(* IEC 61131-3 sources: HappyLearnCodesys/content/softmotion/BasicMotion_DigitalCamSwitch_HighPrecision, 11 files *)

(* ---- GVL_EL2252.st ---- *)
{attribute 'qualified_only'}
VAR_GLOBAL CONSTANT
    /// Maximum number of channels for the EL2252
    NUM_CHANNELS : UDINT := 2;
END_VAR

(* ---- GVL_GVL_EL2252.st ---- *)
END_VAR
{attribute 'qualified_only'}
VAR_GLOBAL CONSTANT
NUM_CHANNELS : UDINT := 2;
/// Maximum number of channels for the EL2252

(* ---- DurationTo32bitEtcTimestamp.st ---- *)
/// Converts duration in seconds to 32bit EtherCAT timestamp in nanoseconds.
FUNCTION DurationTo32bitEtcTimestamp : UDINT
VAR_IN_OUT
    Axis : AXIS_REF_SM3;
	ETCMaster : IODrvEtherCAT;
END_VAR
VAR_INPUT
    duration : LREAL;
END_VAR
VAR
    timestamp64Bit : ULINT;
END_VAR

timestamp64Bit := DurationTo64bitEtcTimestamp(Axis, ETCMaster, duration);
DurationTo32bitEtcTimestamp := TO_UDINT(timestamp64Bit AND 16#FFFF_FFFF);

(* ---- DurationTo64bitEtcTimestamp.st ---- *)
/// Converts duration in seconds to 64bit EtherCAT timestamp in nanoseconds.
FUNCTION DurationTo64bitEtcTimestamp : ULINT
VAR_IN_OUT
    Axis : AXIS_REF_SM3;
	ETCMaster : IODrvEtherCAT;
END_VAR
VAR_INPUT
    duration : LREAL;
END_VAR
VAR
    curTime_ns : ULINT;
	error : SMC_ERROR ;
END_VAR

{IF defined (pou: AXIS_REF_SM3.GetTimestampActValues)}
// GetTimeStampActValues exists for SoftMotion version 4.19.0.0 and higher.
error := Axis.GetTimestampActValues(CurrentActTime=> curTime_ns);
IF error = SMC_NOT_IMPLEMENTED THEN
	// No EtherCAT drive, fall back to default implementation
	curTime_ns := ETCMaster.DCClockReferenceTime;
END_IF
{ELSE}
curTime_ns := ETCMaster.DCClockReferenceTime;
{END_IF}
DurationTo64bitEtcTimestamp := curTime_ns + TO_ULINT(duration*1E9);

(* ---- EventId_GreaterThan.st ---- *)
/// Returns whether the given event Id id1 is greater than the event Id id2.
/// Note that if id2 is not valid, id1 is considered greater.
FUNCTION EventId_GreaterThan : BOOL
VAR_INPUT
    id1 : UDINT;
END_VAR
VAR_IN_OUT CONSTANT
    id2 : EventId;
END_VAR

IF NOT id2.valid THEN
    EventId_GreaterThan := TRUE;
ELSE
    // Greater than check with handling of 32-bit overflows
    EventId_GreaterThan :=
        (id1 > id2.id AND id1 - id2.id < 16#7FFF_FFFF) OR_ELSE
        (id1 < id2.id AND id2.id - id1 > 16#7FFF_FFFF);
END_IF

(* ---- EventId_Init.st ---- *)
FUNCTION EventId_Init
VAR_IN_OUT
    lte : EventId;
END_VAR

lte.id := 0;
lte.valid := FALSE;

(* ---- EventId_Set.st ---- *)
FUNCTION EventId_Set
VAR_IN_OUT
    lte : EventId;
END_VAR
VAR_INPUT
    id : UDINT;
END_VAR

lte.id := id;
lte.valid := TRUE;

(* ---- LogEvent.st ---- *)
FUNCTION LogEvent
VAR_INPUT
    prefix : STRING;
    track : UDINT;
    event : SMC_CAMSWITCH_TOGGLE_EVENT;
    etcTimestamp : ULINT;
    missed : BOOL;
END_VAR

SM0.DoLog(CmpLog.LogClass.LOG_INFO,
    CONCAT(prefix,
    CONCAT(SEL(missed, 'Event tr=', 'MISSED Event tr='),
    CONCAT(TO_STRING(track),
    CONCAT(', sw=',
    CONCAT(TO_STRING(event.SwitchNumber),
    CONCAT(', id=',
    CONCAT(TO_STRING(event.ToggleEventId),
    CONCAT(', v=',
    CONCAT(TO_STRING(event.NewValue),
    CONCAT(', timestamp=',
           TO_STRING(etcTimestamp))))))))))));

(* ---- DigitalCamSwitch_EL2252.st ---- *)
/// This function block shows how to use the output Events from
/// SMC_DigitalCamSwitch_HighPrecision to program a Beckhoff EL2252
/// digital output card.
///
/// The function block assumes that the PDO configuration of the
/// EL2252 contains the outputs to control the two channels
/// and the Feedback input.
/// The PDO values should get mapped to the ``In`` and ``Out``
/// variables of this function block (see the I/O mapping page
/// in the device editor of the EL2252).
///
/// Please note that one track is mapped to one channel of the EL2252 card.
/// The term track and channel are used interchangeably.
FUNCTION_BLOCK DigitalCamSwitch_EL2252
VAR_IN_OUT CONSTANT
    /// The events computed by SMC_DigitalCamSwitch_Forecast.
    Events : SMC_CAMSWITCH_TRACKS_EVENTS;
END_VAR
VAR_IN_OUT
    Axis : AXIS_REF_SM3;
	ETCMaster : IODrvEtherCAT;
END_VAR
VAR_INPUT
    /// Enables the function block.  Enable this function block with the
    /// same signal that enables the SMC_DigitalCamSwitch_HighPrecision
    /// function block.
    Enable : BOOL;
    /// The task interval of the bus task in seconds.
    taskInterval_s : LREAL;
    /// The required inputs of the EL2252.
    In : EL2252_In;
END_VAR
VAR_OUTPUT
    Busy : BOOL ;
    Error : BOOL ;
    /// The outputs, to be mapped to the I/O channels of the EL2252
    Out : EL2252_Out;
    /// Indicates how many events could not be programmed, because the
    /// duration until the event occured was too short (less than
    /// MIN_CYCLES cycles).
    missedCounter : UDINT;
END_VAR
VAR
    state : UDINT;
    EnableOld : BOOL;
    /// Stores for each track the last processed
    /// toggle event id.  This is done to avoid to program
    /// the same switch event twice.
    aLastEventIds : ARRAY[1..GVL_EL2252.NUM_CHANNELS] OF EventId;
END_VAR
VAR_TEMP
    channel : UDINT;
    nextEvents : ARRAY[1..GVL_EL2252.NUM_CHANNELS] OF EL2252_Event;
    eventIdx : UDINT;
    id : UDINT;
    lowestDuration : LREAL := FPU.GetLRealSpecialVal(FPU.ESpecial_FP_Value.PosInf);
    doInputsMatchOutputs : BOOL;
END_VAR
VAR CONSTANT
    EL2252_ACTIVATE_PREPARE : USINT := 0;
    EL2252_ACTIVATE_EVENT : USINT := 3;
    // Time in cycles the output card needs to program an event
    MIN_CYCLES : UDINT := 4;

    STATE_IDLE   : UDINT := 0;
    STATE_INIT : UDINT := 10;
    STATE_CHECK_FOR_EVENT : UDINT := 20;
    STATE_ACTIVATE_EVENT_IN_EL2252 : UDINT := 30;
    STATE_WAIT_UNTIL_THE_INPUTS_MATCH_THE_OUTPUTS : UDINT := 40;
    STATE_ERROR : UDINT := 1000;
END_VAR

IF Enable AND NOT EnableOld THEN
    state := STATE_INIT ;
ELSIF NOT Enable THEN
    state := STATE_IDLE ;
END_IF

CASE state OF
STATE_INIT:
    missedCounter := 0;
    FOR channel := 1 TO GVL_EL2252.NUM_CHANNELS DO
        // Reset stored toggle event id.
        EventId_Init(aLastEventIds[channel]);
    END_FOR
    state := STATE_CHECK_FOR_EVENT;

STATE_CHECK_FOR_EVENT:
    /// Get the next event for each channel.
    FOR channel := 1 TO GVL_EL2252.NUM_CHANNELS DO
        nextEvents[channel].isValid := FALSE;
        nextEvents[channel].activate := FALSE;

        FOR eventIdx := 1 TO Events[channel].numEvents DO
            id := Events[channel].a[eventIdx].ToggleEventId;

            IF EventId_GreaterThan(id, aLastEventIds[channel]) THEN
                IF IsValidDuration(Events[channel].a[eventIdx].Duration) THEN
                    nextEvents[channel].isValid := TRUE;
                    nextEvents[channel].event := Events[channel].a[eventIdx];
                    EXIT;
                ELSE
                    OnMissedEvent(Axis, ETCMaster, channel, Events[channel].a[eventIdx]);
                END_IF
            END_IF
        END_FOR
    END_FOR

    /// Find the event (or events if the events of different channels
    /// have the same duration) with the lowest duration (i.e. the
    /// event that will trigger next).
    FOR channel := 1 TO GVL_EL2252.NUM_CHANNELS DO
        IF nextEvents[channel].isValid THEN
            lowestDuration := MIN(lowestDuration, nextEvents[channel].event.Duration);
        END_IF
    END_FOR

    /// Check which events match the lowestDuration and activate these events.
    FOR channel := 1 TO GVL_EL2252.NUM_CHANNELS DO
        IF nextEvents[channel].isValid AND lowestDuration = nextEvents[channel].event.Duration THEN
            nextEvents[channel].activate := TRUE;
        END_IF
    END_FOR

    /// Write the outputs
    FOR channel := 1 TO GVL_EL2252.NUM_CHANNELS DO
        IF nextEvents[channel].activate THEN
            EventId_Set(aLastEventIds[channel], nextEvents[channel].event.ToggleEventId);

            Out.activate := EL2252_ACTIVATE_PREPARE;
            Out.startTime := DurationTo64bitEtcTimestamp(Axis, ETCMaster, nextEvents[channel].event.Duration);
            Out.channels[channel].output := nextEvents[channel].event.NewValue;

			LogEvent(
                prefix:= 'EL2252: ',
                track:= channel,
                event:= nextEvents[channel].event,
                etcTimestamp:= Out.startTime,
                missed:= FALSE);

            state := STATE_ACTIVATE_EVENT_IN_EL2252;
        END_IF
    END_FOR

STATE_ACTIVATE_EVENT_IN_EL2252:
    Out.activate := EL2252_ACTIVATE_EVENT;

    state := STATE_WAIT_UNTIL_THE_INPUTS_MATCH_THE_OUTPUTS;

STATE_WAIT_UNTIL_THE_INPUTS_MATCH_THE_OUTPUTS:
    doInputsMatchOutputs := TRUE;
    FOR channel := 1 TO GVL_EL2252.NUM_CHANNELS DO
        doInputsMatchOutputs :=
            doInputsMatchOutputs
            AND In.channels[channel].output = Out.channels[channel].output
            AND In.channels[channel].triState = Out.channels[channel].triState;
    END_FOR

    IF doInputsMatchOutputs THEN
        state := STATE_CHECK_FOR_EVENT;
    END_IF
END_CASE

IF IsBusy() THEN
    /// Check for events that will be missed.
    FOR channel := 1 TO GVL_EL2252.NUM_CHANNELS DO
        FOR eventIdx := 1 TO Events[channel].numEvents DO
            id := Events[channel].a[eventIdx].ToggleEventId;

            IF EventId_GreaterThan(id, aLastEventIds[channel])
               AND NOT IsValidDuration(Events[channel].a[eventIdx].Duration)
            THEN
                OnMissedEvent(Axis, ETCMaster, channel, Events[channel].a[eventIdx]);
            END_IF
        END_FOR
    END_FOR
END_IF

OnExit();

(* ---- DigitalCamSwitch_EL2258.st ---- *)
/// This function block shows how to use the output Events from
/// SMC_DigitalCamSwitch_HighPrecision to program a Beckhoff EL2258
/// digital output card.
///
/// The function block assumes that the PDO configuration of the
/// EL2258 contains two channels, each with at least 2 events.
/// The members of the arrays ChannelsOut and ChannelsIn must
/// be mapped to the I/O channels of the EL2258 device in the
/// I/O mapping page of the device editor.
///
/// Please note that one track is mapped to one channel of the EL2258 card.
/// The term track and channel are used interchangeably.
FUNCTION_BLOCK DigitalCamSwitch_EL2258
VAR_IN_OUT CONSTANT
    /// The events computed by SMC_DigitalCamSwitch_Forecast.
    Events : SMC_CAMSWITCH_TRACKS_EVENTS;
END_VAR
VAR_IN_OUT
    Axis : AXIS_REF_SM3;
	ETCMaster : IODrvEtherCAT;
END_VAR
VAR_INPUT
    /// Enables the function block.  Enable this function block with the
    /// same signal that enables the SMC_DigitalCamSwitch_HighPrecision
    /// function block.
    Enable : BOOL;
    /// The task interval of the bus task in seconds.
    taskInterval_s : LREAL;
END_VAR
VAR_OUTPUT
    Busy : BOOL ;
    Error : BOOL ;

    /// The output channels, to be mapped to the I/O channels of the EL2258
    ChannelsOut : ARRAY[1..NUM_CHANNELS] OF EL2258_OutChannel ;
    /// The input channels, to be mapped to the I/O channels of the EL2258
    ChannelsIn : ARRAY[1..NUM_CHANNELS] OF EL2258_InChannel ;

	/// Indicates how many events could not be programmed, because the
	/// duration until the event occured was too short (less than
	/// MIN_CYCLES cycles).
    missedCounter : UDINT;
END_VAR
VAR
    state : UDINT;
    EnableOld : BOOL;

    /// Stores for each track the last processed
    /// toggle event id.  This is done to avoid to program
    /// the same switch event twice.
    aLastEventIds : ARRAY[1..NUM_CHANNELS] OF EventId;
END_VAR
VAR_TEMP
    channel : UDINT;
    id : UDINT;
    i : UDINT;
    event : POINTER TO SMC_CAMSWITCH_TOGGLE_EVENT;
    etcTimestamp : UDINT;
    nEvents : UDINT;
    missed : BOOL;
END_VAR
VAR CONSTANT
    NUM_CHANNELS : UDINT := 2;
    // Time in cycles the output card needs to program an event
    MIN_CYCLES : UDINT := 6;

    STATE_IDLE   : UDINT := 0;
    STATE_INIT_0 : UDINT := 10;
    STATE_INIT_1 : UDINT := 20;
    STATE_ACTIVE : UDINT := 30;
    STATE_ERROR  : UDINT := 1000;
END_VAR

IF Enable AND NOT EnableOld THEN
    state := STATE_INIT_0 ;
ELSIF NOT Enable THEN
    state := STATE_IDLE ;
END_IF

CASE state OF
STATE_INIT_0:
    missedCounter := 0;
    FOR channel := 1 TO NUM_CHANNELS DO
        // Reset ouput buffer of the terminal EL2258
        ChannelsOut[channel].OutputBufferReset := TRUE;

        // Reset stored toggle event id.
        EventId_Init(aLastEventIds[channel]);
    END_FOR
    state := STATE_INIT_1;

STATE_INIT_1:
    FOR channel := 1 TO NUM_CHANNELS DO
        ChannelsOut[channel].OutputBufferReset := FALSE;
    END_FOR
    state := STATE_ACTIVE;

STATE_ACTIVE:
    FOR channel := 1 TO NUM_CHANNELS DO
        // Previous events already procesed by the output card?
        IF ChannelsIn[channel].OutputOrderFeedback = ChannelsOut[channel].OutputOrderCounter THEN
            // Program the next up to five events for this channel
            nEvents := 0;
            i := 1;
            WHILE i <= Events[channel].numEvents AND nEvents < 5 DO
                event := ADR(Events[channel].a[i]);
                id := event^.ToggleEventId;

                // Only process events with an Id greater then the last processed
                // Id for this switch number.
                IF EventId_GreaterThan(id, aLastEventIds[channel]) THEN
                    etcTimestamp := DurationTo32bitEtcTimestamp(Axis, ETCMaster, event^.Duration);

                    IF event^.Duration < MIN_CYCLES * taskInterval_s THEN
                         // Less then MIN_CYCLES left until the switch occurs.
                         // There is not enough time to program the switch.
                         missedCounter := missedCounter + 1 ;
                         missed := TRUE;
                    ELSE
                         missed := FALSE;
						 ChannelsOut[channel].OutputEventState[nEvents] := event^.NewValue;
						 ChannelsOut[channel].OutputEventTime[nEvents] := etcTimestamp;

						 nEvents := nEvents + 1 ;
                    END_IF

					EventId_Set(aLastEventIds[channel], id);
                    LogEvent(
						prefix:= 'EL2258: ',
                        track:= channel,
                        event:= event^,
                        etcTimestamp:= etcTimestamp,
                        missed:= missed);
                END_IF

                i := i + 1;
            END_WHILE

            IF nEvents > 0 THEN
                ChannelsOut[channel].NoOfOutputEvents := TO_USINT(nEvents);

                // Trigger Multi-Timestamp scheduling
                ChannelsOut[channel].OutputOrderCounter := ChannelsOut[channel].OutputOrderCounter + 1;
            END_IF
        END_IF
    END_FOR
END_CASE

OnExit();

(* ---- Main.st ---- *)
PROGRAM Main
VAR
    pw : MC_Power;
    mv : MC_MoveVelocity := (Velocity:= 180, Acceleration:= 3600, Deceleration:= 3600, Jerk:= 36000);

    aSwitches : ARRAY[0..7] OF MC_CAMSWITCH_TR := [
        (TrackNumber:= 1,
         FirstOnPosition:= 20,
         LastOnPosition:= 90,
         AxisDirection:= 1,  // positive
         CamSwitchMode:= 0), // position based
        (TrackNumber:= 1,
         FirstOnPosition:= 180,
         LastOnPosition:= 270,
         AxisDirection:= 1,  // positive
         CamSwitchMode:= 0), // position based
        (TrackNumber:= 2,
         FirstOnPosition:= 30,
         LastOnPosition:= 90,
         AxisDirection:= 1,  // positive
         CamSwitchMode:= 0), // position based
        (TrackNumber:= 2,
         FirstOnPosition:= 190,
         LastOnPosition:= 270,
         AxisDirection:= 1,  // positive
         CamSwitchMode:= 0)]; // position based

    switches : MC_CAMSWITCH_REF := (
            NoOfSwitches := 4,
            CamSwitchPtr:= ADR(aSwitches));

    tracks : MC_TRACK_REF :=[
            (OnCompensation:= -0.1,
             OffCompensation:= 0.1),
            (OnCompensation:= 0.05,
             OffCompensation:= -0.05)];

    setForecast : SMC_SetForecast := (ForecastDuration:= 0.15);

    dcs : SMC_DigitalCamSwitch_HighPrecision;
    dcs_el2258 : DigitalCamSwitch_EL2258;
	dcs_el2252 : DigitalCamSwitch_EL2252;

    state : UDINT ;
END_VAR

CASE state OF
0:
    setForecast.Execute := TRUE;
    IF setForecast.Done THEN
        state := state + 10;
    END_IF

10:
    pw.Enable := TRUE;
    pw.bRegulatorOn := TRUE;
    pw.bDriveStart := TRUE;

    IF pw.Status THEN
        state := state + 10;
    END_IF

20:
    IF EtherCAT_Master_SoftMotion.GetBusState() = DED.BUS_STATE.RUNNING THEN
        state := state + 10;
    END_IF

30:
    mv.Execute := TRUE;
    dcs.Enable := TRUE;
    dcs_el2258.Enable := TRUE;
	dcs_el2252.Enable := TRUE;
END_CASE

pw(Axis:= Drive);
mv(Axis:= Drive);
setForecast(Axis:= Drive);
dcs(Axis:= Drive, Switches:= switches, TrackOptions:= tracks);
dcs_el2258(
    Events:= dcs.Events,
    Axis:= Drive,
	ETCMaster:= EtherCAT_Master_SoftMotion,
    taskInterval_s:= Drive.fTaskCycle);
dcs_el2252(
    Events:= dcs.Events,
    Axis:= Drive,
	ETCMaster:= EtherCAT_Master_SoftMotion,
    taskInterval_s:= Drive.fTaskCycle);
